(*~
	<docu>
		<summary>
			Data task is a remote task  <see cref="PlcDocu.TcoCore.RemoteTask"/> with a paramater. 	
		</summary>	
		<param name="_identifier">The Identifier, ID  of an entity on which a CRUD operation should be executed</param>
		<remarks>Inxton is required for this feature to work</remarks>		
	</docu>	
~*)
FUNCTION_BLOCK TcoDataTask EXTENDS TcoCore.TcoRemoteTask
VAR
	(*~
	<docu>
		<summary>
			The Identifier, ID  of an entity on which a CRUD operation should be executed. 	
		</summary>						
	</docu>	
	~*)
    _identifier : STRING(255);
END_VAR

SUPER^();

METHOD PUBLIC FB_init : BOOL
VAR_INPUT
	bInitRetains : BOOL; // if TRUE, the retain variables are initialized (warm start / cold start)
	bInCopyCode : BOOL;  // if TRUE, the instance afterwards gets moved into the copy code (online change)
	ParentObject : TcoCore.ITcoObject;	
END_VAR
END_METHOD

(*~
	<docu>
		<summary>
			Executes CRUD operation on data entry with given identifier. 	
		</summary>			
		<remarks>Inxton is required for this feature to work</remarks>		
	</docu>	
~*)
METHOD WithId : REFERENCE TO TcoDataTask
VAR_INPUT
	(*~
	<docu>
		<summary>
			The Identifier, ID  of an entity on which a CRUD operation should be executed. 	
		</summary>						
	</docu>	
	~*)
	inIdentifier : STRING(254);
END_VAR
THIS^._identifier := inIdentifier;
WithId REF= THIS^;
END_METHOD

END_FUNCTION_BLOCK

(* stored: Version 1.1.0.1, ProductVersion 3.1.4024.12
   POU TcoDataTask: Id {d746b7c0-aeef-0bb8-363a-a8b912d682b6}, SpecialFunc None
   Method FB_init: Id {03c5aeaf-9a88-0e65-2886-43aec8e1a787}
   Method WithId: Id {d8ebbe97-9c86-0568-17c4-bcc05d378bb1} *)
